// TIA Portal project "3M -1" (V16)

(* hardware
DEVICE "S7-1200 station_1"  S7-1200 Station
   slot 0: "Rack_0"  S7-1200 Rack  Rack  V1.0
   slot 1: "PLC_1"  CPU 1212C AC/DC/Rly  6ES7 212-1BE40-0XB0  V4.0
*)

// ===== PLC "PLC_1"  CPU 1212C AC/DC/Rly =====

VAR_GLOBAL   // PLC tag table "Default tag table"
   "K1" AT %Q0.0 : Bool;
   "stop1" AT %I0.4 : Bool;
   "k2" AT %Q0.1 : Bool;
   "X" AT %M0.0 : Bool;
   "K3" AT %Q0.2 : Bool;
   "start1" AT %I0.2 : Bool;
   "T1 tag" AT %M0.1 : Bool;
   "T2 tag" AT %M0.2 : Bool;
   "T3 tag" AT %M0.3 : Bool;
   "Y" AT %M1.0 : Bool;
   "Z" AT %M1.2 : Bool;
   "Tag_1" AT %I0.3 : Bool;
END_VAR

// folder: System blocks/Program resources

DATA_BLOCK "T1"   // DB2
{ S7_Optimized_Access := 'TRUE' }
AUTHOR : Simatic
FAMILY : IEC
NAME : IEC_TMR
VERSION : 1.0
// stored: InstanceOfName IEC_TIMER
"IEC_TIMER"
BEGIN
END_DATA_BLOCK

DATA_BLOCK "T2"   // DB3
{ S7_Optimized_Access := 'TRUE' }
AUTHOR : Simatic
FAMILY : IEC
NAME : IEC_TMR
VERSION : 1.0
// stored: InstanceOfName IEC_TIMER
"IEC_TIMER"
BEGIN
END_DATA_BLOCK

DATA_BLOCK "T3"   // DB4
{ S7_Optimized_Access := 'TRUE' }
AUTHOR : Simatic
FAMILY : IEC
NAME : IEC_TMR
VERSION : 1.0
// stored: InstanceOfName IEC_TIMER
"IEC_TIMER"
BEGIN
END_DATA_BLOCK

// folder: (top level)

ORGANIZATION_BLOCK "Main"   // OB1, LAD, ProgramCycle
TITLE = "Main Program Sweep (Cycle)"
{ S7_Optimized_Access := 'TRUE' }
VERSION : 0.1
   VAR_INPUT
      Initial_Call : Bool;   // Initial call of this OB
      Remanence : Bool;   // =True, if remanent data are available
   END_VAR
BEGIN

REGION Network 1: start
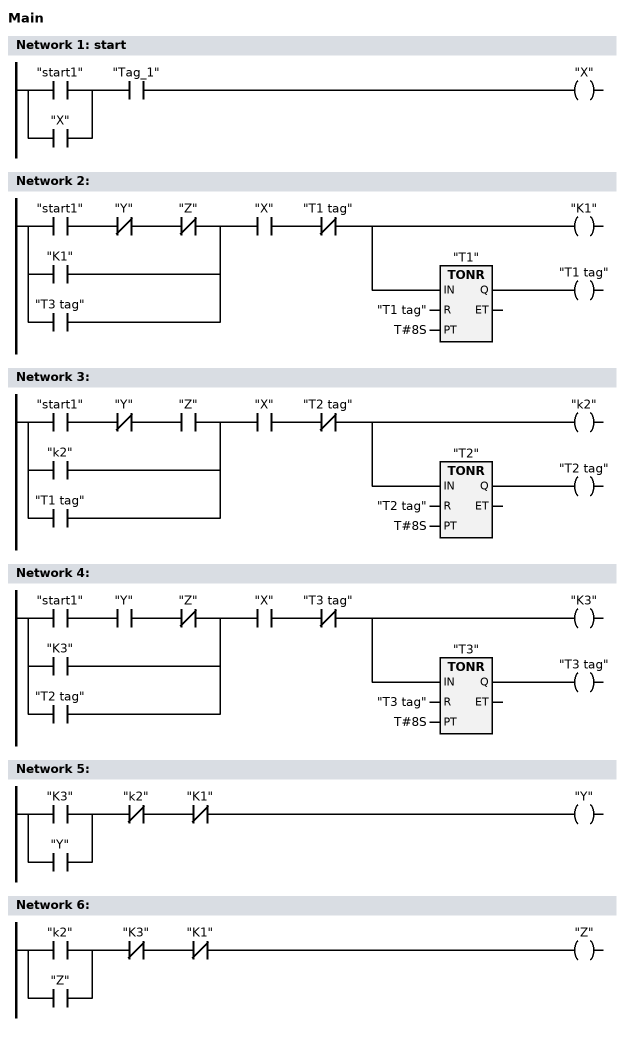
   RUNG wire#powerrail
      Contact( "start1" )
      wire#w1
      Contact( "Tag_1" )
      Coil( "X" )
   END_RUNG
   RUNG wire#powerrail
      Contact( "X" )
   END_RUNG wire#w1
   // the same network as SCL:
   "X" := ("start1" OR "X") AND "Tag_1";
END_REGION

REGION Network 2
   "K1" := (("start1" AND NOT "Y" AND NOT "Z") OR "K1" OR "T3 tag") AND "X" AND NOT "T1 tag";
   "T1".TONR(IN := "K1", R := "T1 tag", PT := T#8S);
   "T1 tag" := "T1".Q;
END_REGION

REGION Network 3
   "k2" := (("start1" AND NOT "Y" AND "Z") OR "k2" OR "T1 tag") AND "X" AND NOT "T2 tag";
   "T2".TONR(IN := "k2", R := "T2 tag", PT := T#8S);
   "T2 tag" := "T2".Q;
END_REGION

REGION Network 4
   "K3" := (("start1" AND "Y" AND NOT "Z") OR "K3" OR "T2 tag") AND "X" AND NOT "T3 tag";
   "T3".TONR(IN := "K3", R := "T3 tag", PT := T#8S);
   "T3 tag" := "T3".Q;
END_REGION

REGION Network 5
   RUNG wire#powerrail
      Contact( "K3" )
      wire#w1
      I_Contact( "k2" )
      I_Contact( "K1" )
      Coil( "Y" )
   END_RUNG
   RUNG wire#powerrail
      Contact( "Y" )
   END_RUNG wire#w1
   // the same network as SCL:
   "Y" := ("K3" OR "Y") AND NOT "k2" AND NOT "K1";
END_REGION

REGION Network 6
   RUNG wire#powerrail
      Contact( "k2" )
      wire#w1
      I_Contact( "K3" )
      I_Contact( "K1" )
      Coil( "Z" )
   END_RUNG
   RUNG wire#powerrail
      Contact( "Z" )
   END_RUNG wire#w1
   // the same network as SCL:
   "Z" := ("k2" OR "Z") AND NOT "K3" AND NOT "K1";
END_REGION
END_ORGANIZATION_BLOCK